PROGRAM JIG
VAR
	BasketA_Plus	: BOOL;
	BasketA_Minus	: BOOL;
	BasketB_Plus	: BOOL;
	BasketB_Minus	: BOOL;
	MAX_FG_ON_BASKET : UINT := 15;
END_VAR

IF AUTO_MODE.AutoMode THEN
	RETURN;
END_IF

GVL.JIGA_Release := NOT GVL.JIGA_Clamp;
GVL.JIGB_Release := NOT GVL.JIGB_Clamp;
GVL.JIGC_Release := NOT GVL.JIGC_Clamp;

IF BasketA_Plus THEN
	GVL.Basket_A_Counter := GVL.Basket_A_Counter + 1;
	IF GVL.Basket_A_Counter > MAX_FG_ON_BASKET THEN
		GVL.Basket_A_Counter := 0 ;
	END_IF
	BasketA_Plus := FALSE;
END_IF

IF BasketA_Minus THEN
	GVL.Basket_A_Counter := GVL.Basket_A_Counter - 1;
	IF GVL.Basket_A_Counter < 0 THEN
		GVL.Basket_A_Counter := MAX_FG_ON_BASKET;
	END_IF
	BasketA_Minus := FALSE;
END_IF

IF BasketB_Plus THEN
	GVL.Basket_B_Counter := GVL.Basket_B_Counter + 1;
	IF GVL.Basket_B_Counter > MAX_FG_ON_BASKET THEN
		GVL.Basket_B_Counter := 0 ;
	END_IF
	BasketB_Plus := FALSE;
END_IF

IF BasketB_Minus THEN
	GVL.Basket_B_Counter := GVL.Basket_B_Counter - 1;
	IF GVL.Basket_B_Counter < 0 THEN
		GVL.Basket_B_Counter := MAX_FG_ON_BASKET;
	END_IF
	BasketB_Minus := FALSE;
END_IF

END_PROGRAM

(* stored: Version 1.1.0.1, ProductVersion 3.1.4024.12
   POU JIG: Id {12d6e6ee-325e-4362-970c-94c78e2dc5b6}, SpecialFunc None *)
